// TwinCAT 3 PLC project SimulationPLC
// ProgramVersion: 3.1.4023.0
// libraries:
//   Tc2_Standard, * (Beckhoff Automation GmbH)
//   Tc2_System, * (Beckhoff Automation GmbH)
//   Tc3_Module, * (Beckhoff Automation GmbH)
// project tree:
//   GVLs/Communications/ DataExchange.TcGVL
//   / PlcTask.TcTTO
//   POUs/ MAIN.TcPOU

CONFIGURATION SimulationPLC
    RESOURCE PLC ON TwinCAT3
        TASK PlcTask(INTERVAL := T#10ms, PRIORITY := 20);
        PROGRAM MAIN WITH PlcTask : MAIN;
    END_RESOURCE
END_CONFIGURATION

// ---- GVLs/Communications/DataExchange.TcGVL
{attribute 'qualified_only'}
VAR_GLOBAL
	spawnRate: REAL := 2;
	boxSpeed: REAL := 3;
	runBelt: BOOL := TRUE;
	autoDirection: BOOL := TRUE;
	direction: DINT := 0; //0 = left , else = right
END_VAR

// ---- POUs/MAIN.TcPOU
PROGRAM MAIN
VAR
	boxSpeed : REAL;
	spawnRate: REAL;
	runBelt: BOOL;
	autoDirection: BOOL;
	direction: DINT; //0 = left , else = right
END_VAR

boxSpeed := DataExchange.boxSpeed;
spawnRate := DataExchange.spawnRate;
runBelt := DataExchange.runBelt;
autoDirection := DataExchange.autoDirection;
direction := DataExchange.direction;

END_PROGRAM
